{attribute 'GeneratedUsingTerminal: BK1120-0000-0019'}
{attribute addProperty BoxType "BK1120-0000-0019"}
{attribute addProperty Id "Term_379_KL1002KL1002_BB38DA8F0"}
{attribute addProperty CRC "2490385770"}
{attribute addProperty Size "0"}
TYPE A_0006_BK1120_0000_0019_9470456A EXTENDS BK1120_A2FCADE7 :
STRUCT
	{attribute addProperty Name "Term_379_KL1002"}
	Term_379_KL1002 : KL1002_BB38DA8F;
END_STRUCT
END_TYPE

(* stored: Version 1.2.0.0, ProductVersion 3.1.4024.9
   DUT A_0006_BK1120_0000_0019_9470456A: Id {f2a2ae1c-9ce5-46e2-bcc6-419cfde0851b} *)
